FUNCTION_BLOCK ABSTRACT FB_SimStation IMPLEMENTS IStation
VAR_INPUT
END_VAR
VAR_OUTPUT
END_VAR
VAR
	bPartPresent				AT %I* : BOOL;
	bReady						: BOOL;
	bFaulted					: BOOL;
	
	StationState				: E_SimStationState;
	pPartStatus					: POINTER TO ST_PartStatus;
	tmrDelay					: TON;
END_VAR

METHOD PROTECTED ABSTRACT DoWork : BOOL
VAR_INPUT
END_VAR
END_METHOD

METHOD Execute : PVOID
CASE StationState OF
	
	E_SimStationState.IDLE:
		
		tmrDelay(IN:=bPartPresent, PT:=T#100MS);
		
		IF bPartPresent THEN
			bReady := FALSE;
			IF tmrDelay.Q THEN
				StationState := E_SimStationState.WORKING;
			END_IF
		ELSE
			bReady := TRUE;
		END_IF
		
	E_SimStationState.WORKING:
		
		bReady := FALSE;
		
		IF DoWork() THEN
			StationState := E_SimStationState.DONE;
		END_IF
	
	E_SimStationState.DONE:
	
		bReady := TRUE;
		
		IF NOT bPartPresent THEN
			UpdatePartStatus();
			StationState := E_SimStationState.IDLE;
		END_IF
		
END_CASE
END_METHOD

PROPERTY Faulted : BOOL
GET
Faulted := bFaulted;
END_GET
END_PROPERTY

PROPERTY PartPresent : BOOL
GET
PartPresent := bPartPresent;
END_GET
END_PROPERTY

PROPERTY PartStatus : POINTER TO ST_PartStatus
SET
pPartStatus := PartStatus;
END_SET
END_PROPERTY

PROPERTY Ready : BOOL
GET
Ready := bReady;
END_GET
END_PROPERTY

METHOD PROTECTED ABSTRACT UpdatePartStatus : PVOID
VAR_INPUT
END_VAR
END_METHOD

END_FUNCTION_BLOCK

(* stored: Version 1.1.0.1, ProductVersion 3.1.4024.12
   POU FB_SimStation: Id {d0a3379f-7809-46be-8a25-c7aab289bc1a}, SpecialFunc None
   Method DoWork: Id {e5a556de-42b2-42cf-b082-085ffc0c5809}
   Method Execute: Id {22f70b89-6c8b-41b6-85f0-a0877a445ffc}
   Property Faulted: Id {bba4ac03-8451-4afa-850d-3d9f30cc03cc}
   Get Get: Id {d888a9d9-d513-462c-a1d9-d769c3a3cf57}
   Property PartPresent: Id {93b29da4-32df-4649-80a2-9cd532bebaff}
   Get Get: Id {f6607e3c-3f2a-4515-b47c-0c118b440b03}
   Property PartStatus: Id {2b5862fc-d124-4970-8444-6d63caf7fb86}
   Set Set: Id {4241aacb-02f9-4f86-8c79-0e8cb03aaabd}
   Property Ready: Id {8d558544-163c-40c3-b4b3-67bbf215193b}
   Get Get: Id {14a9f377-1a11-46ad-991d-5dadbd5a3997}
   Method UpdatePartStatus: Id {509a9894-fb9e-425c-aff0-b182d101e493} *)
